FUNCTION_BLOCK "GCS7_E_PressureRange"	// FB 16
TITLE = PressureRange
//  
//COPYRIGHT:    (C) 1996  BUHLER AG, CH-9240 UZWIL, SWITZERLAND
//
//PRODUCT:      GCS7
//
//TITLE:        Pressure Range
//
//-------------------------------------------------------------------------
//
//IDENT:        AUTHOR:             DEPT:                       DATE:
//
//FB16.4.1      A. Egli             CT3                         09-Mar-2004
//              PCDirect Control: CmdReportOn,CmdReportOff=Bit14
//FB16.4.0      A. Egli             CT3                         17-Jun-2002
//              New Release with one block 
//FB16.2.2      S. Kalberer         CT3                         16-Oct-2000
//              LOG-entry corrected: SPN -> SPBN
//FB16.2.1      A. Egli             CT3                         08-Mai-2000
//              Local: StOverP --> StMinP
//              Set alarm horn by rising edge OutNoMinP
//FB16.2B       A. Egli             CT3                         23-Nov-1999
//              Message Nr StCtoOverP
//FB16.2A       A. Egli             CT3                         04-Mai-1998
//              StFault = StCode 32
//FB16.1A       S. Kalberer         AEE61                       10-Jul-1997
//              1st Release in S7
//
//-------------------------------------------------------------------------
//
//PURPOSE:      MANUAL : see [PRAENMAN]
//
//RESTRICTIONS: S7
//              ACCU2: Pointer to dynamic datas of the element
//              ACCU1: Pointer to parameter datas of the element
//
//-------------------------------------------------------------------------
//=======================================================
//Log Message: 
//------------------------------------------------------
// 0  normal pressure  
// 1  high pressure
// 2  over pressure
// 3  no minimum pressure
// 9  fault cancelled
// 10 fault
//
//=======================================================
//StCode:  State               
//------------------------------------------------------
//32  StFault             
// 1  StMinP              
//41  StMinP.HWStop       
//51  StMinP.DPFault      
// 3  StNormalP           
//43  StNormalP.HWStop    
//53  StNormalP.DPFault   
// 4  StCtoOverP          
//44  StCtoOverP.HWStop   
//54  StCtoOverP.DPFault  
// 5  StOverP             
//45  StOverP.HWStop      
//55  StOverP.DPFault     
// 6  StNormalP.Warning  
//
//
//
AUTHOR : EA
FAMILY : GCS7LL
NAME : PRang
VERSION : 4.1
VAR
  StCode : INT ;	//Element state code
  InMonMinP : BOOL ;	//Monitoring the minimum pressure
  spare0201 : BOOL ;
  spare0202 : BOOL ;
  spare0203 : BOOL ;
  spare0204 : BOOL ;
  spare0205 : BOOL ;
  InpMin : BOOL ;	//Digital input: Value <= min
  InpMax : BOOL ;	//Digital input: Value >= max
  spare0300 : BOOL ;
  spare0301 : BOOL ;
  spare0302 : BOOL ;
  CmdFaultReset : BOOL ;	//Command to reset fault
  InLocal : BOOL ;	//1= Local mode (no fault by Over Pressure)
  spare0305 : BOOL ;
  InReport : BOOL ;	//Report of all state transition
  spare0307 : BOOL ;
  InHWStop : BOOL ;	//HW stop is detected, no fault
  InDPFault : BOOL ;	//DP-Fault is detected, no fault
  OutNoMinP : BOOL ;	//Warning no minimum pressure
  spare0403 : BOOL ;
  spare0404 : BOOL ;
  spare0405 : BOOL ;
  spare0406 : BOOL ;
  spare0407 : BOOL ;
  StMinP : BOOL ;	//Value <= Minimum
  StNormalP : BOOL ;	//Value in Range Minimum to Maximum
  StOverP : BOOL ;	//Value >= Maximum (only in local mode)
  StCtoOverP : BOOL ;	//Value >= Maximum, delay time is active
  StFault : BOOL ;	//Element has a fault
  OutAlarmNrLog : INT ;	//Last textnumber send to log
  Par : STRUCT
   ParObjectNo : INT ;	//Is used for communication with PC, e.g. for message
   ParMsgType : INT ;	//Is used for message (translation of state)
   ParHornCode : INT ;	//Is used by horn module
   ParLogOff : BOOL ;	//Report is off
   ParDelayChange : INT ;	//t0, maximum time until state changes to StCtoOverP
   ParDelayMin : INT ;	//t1, maximum time until state changes to StMinP
   ParDelayMax : INT ;	//t2, maximum time until state changes to StOverP or StFault
   ParMonMinP : INT ;	//t3, if InMonMinP: maximum time to be out of MinP until OutNoMinP
   OutMonTime : INT ;	//Actual value monitoring time t3
   OutDelayMinTime : INT ;	//Actual value delay time t1
   OutDelayMaxTime : INT ;	//Actual value delay time t0,t2
  END_STRUCT ;
END_VAR
VAR_TEMP
  tmpLOGvalue : WORD ;	//LOG value
  tmpLenDyn : DINT ;
  tmpReport : BOOL ;	//Global LOG all
  tmpDelayOver : BOOL ;	//Delay time is over
  tmpLocal : BOOL ;
END_VAR
BEGIN
NETWORK
TITLE =  Start Global
      L     30;
      T     #tmpLenDyn;	// Length Dynamic datas
NETWORK
TITLE = PC Control
//=== Test Object number =====================
      L     "SYS_DirectCtrlDB".PC.ObjectNo;	//PCControl.ObjectNo
      L     #Par.ParObjectNo;	//Input ObjectNo
      <>I;
      JC    Ctrl;
//=== Test OType      ========================
      L     1016;	//Input object type
      L     "SYS_DirectCtrlDB".PC.ObjectType;	//PCControl.ObjectType
      <>I;
      JC    Ctrl;
//=== Test Handshake =========================
      A     "SYS_DirectCtrlDB".PC.Hsk.FExamine;	// Handshake.FExamine
      JC    pExa;
      A     "SYS_DirectCtrlDB".PC.Hsk.FDefineCmd;	// Handshake.FDefineCmd
      JC    pCmd;
      A     "SYS_DirectCtrlDB".PC.Hsk.FDefinePara;	// Handshake.FDefinePara
      JC    pPar;
pIni: L     2;	// FcInit
      UC    "SYS_DirectCtrl";
      JU    Ctrl;
// Write parameter 
pPar: LAR1  P#DBX 58.0;
      L     P##Par;
      L     DW#16#FFFFF;
      AD;
      +AR1;
      L     DBW [AR1,P#8.0];
      T     #Par.ParDelayChange;
      L     DBW [AR1,P#10.0];
      T     #Par.ParDelayMin;
      L     DBW [AR1,P#12.0];
      T     #Par.ParDelayMax;
      L     DBW [AR1,P#14.0];
      T     #Par.ParMonMinP;
// Write new commands from PC to Interface object
pCmd: A     "SYS_DirectCtrlDB".PC.Cmd1[11];	// CmdFaultReset
      S     #CmdFaultReset;
      A     "SYS_DirectCtrlDB".PC.Cmd1[14];	// CmdReportOn    [4.1]
      S     #InReport;
      A     "SYS_DirectCtrlDB".PC.Cmd2[14];	// CmdReportOff   [4.1]
      R     #InReport;
      JU    pIni;
pExa: TAR2;	// Address Dynamic datas
      T     "SYS_DirectCtrlDB".GC.InDynAddr;	// -->PCControl.GC.InDynAddr
      L     #tmpLenDyn;	// Length Dynamic datas
      T     "SYS_DirectCtrlDB".GC.InDynLen;	// -->PCControl.GC.InDynLen
      L     0;
      T     "SYS_DirectCtrlDB".GC.InParaAddr;	// -->PCControl.GC.InParaAddr
      T     "SYS_DirectCtrlDB".GC.InParaLen;	// -->PCControl.GC.InParaLen
      L     1;	// Code FcExamine
      UC    "SYS_DirectCtrl";
      L     10;	//Revision
      T     "SYS_DirectCtrlDB".GC.Revision;
NETWORK
TITLE =  All State Init
//===Global Group Orders===
//---Report is on---
Ctrl: O     "GCS7_Gr_OutReportAll";	//---Global OutReportAll
      O     #InReport;
      =     #tmpReport;
      A     #InLocal;
      O     #InHWStop;
      O     #InDPFault;
      =     #tmpLocal;
// Monitoring
//---Condition to start monitoring time:  Monitoring is on
      A     #InMonMinP;
      AN    #StMinP;	// State minimum pressure
      JC    MO2;
      R     #OutNoMinP;
      L     #Par.ParMonMinP;	// Set monitoring time
      T     #Par.OutMonTime;
      JU    STAT;
//---Condition for monitoring
MO2:  A     #OutNoMinP;	// Monitoring output
      JC    STAT;
      AN    "GCS7_Gr_OutTick200ms";	//Gr.OutTick200ms
      L     #Par.OutMonTime;
      JC    MO3;
      +     -2;	// Decrement all 200ms
      T     #Par.OutMonTime;
MO3:  L     0;
      >I;	// Check monitoring time t3 over
      JC    STAT;
      S     #OutNoMinP;	// set monitoring output
      S     "GCS7_Gr_InFaultFlag";	// InFaultFlag
      CALL  "SYS_Horn_Code" (
           FcCode                   := 1,
           ParObjectType            := 1016,
           ParObjectNo              := #Par.ParObjectNo,
           ParHornCode              := #Par.ParHornCode);
      JU    LOG3;
NETWORK
TITLE = States
STAT: A     #StMinP;	//===State machine===
      JC    MP;
      A     #StNormalP;
      JC    NP;
      A     #StCtoOverP;
      JC    COP;
      A     #StOverP;
      JC    OP;
      A     #StFault;
      JC    FLT;
      S     #StMinP;	//Initialise: goto StMinP
NETWORK
TITLE = StMinP
MP:   A     #InpMin;	//---Condition for StMinP
      AN    #InpMax;
      JC    SAVE;
      R     #StMinP;	//---Transition --> StNormal
      S     #StNormalP;
      L     #Par.ParDelayChange;
      T     #Par.OutDelayMaxTime;
      JU    LOG1;
NETWORK
TITLE = StNormalP
//Logic
//---Condition for StCtoOverP
NP:   A     #InpMax;
      JC    NPJ1;
      L     #Par.ParDelayChange;
      T     #Par.OutDelayMaxTime;
//---Condition for StNormalP
      A     #InpMin;
      R     #StNormalP;
      S     #StMinP;
      JU    SAVE;
NPJ1: L     #Par.OutDelayMaxTime;
      AN    "GCS7_Gr_OutTick200ms";	//Gr.OutTick200ms
      JC    NPJ2;
      +     -2;	// Decrement all 0.2s
      T     #Par.OutDelayMaxTime;
NPJ2: L     0;
      >I;
      JC    SAVE;
//---Transition --> StCtoOverP
      R     #StNormalP;
      S     #StCtoOverP;
      L     #Par.ParDelayMax;
      T     #Par.OutDelayMaxTime;
      L     #Par.ParDelayMin;
      T     #Par.OutDelayMinTime;
      JU    LOG1;
NETWORK
TITLE = StCtoOverP
//---Condition for StCtoOverP
COP:  AN    "GCS7_Gr_OutTick200ms";	//Gr.OutTick200ms
      L     #Par.OutDelayMaxTime;
      JC    COP1;
      +     -2;	// Decrement all 0.2s
      T     #Par.OutDelayMaxTime;
COP1: L     0;
      >I;
      JC    COPM;
//---Transition --> StFault
      AN    #tmpLocal;
      R     #StCtoOverP;
      JC    xxS4;
//---Transition --> StOverP
      R     #StCtoOverP;
      S     #StOverP;
      JU    LOG1;
//---Condition for StMinP
//Condition delay time minimum
COPM: A     #InpMin;
      AN    #InpMax;
      JC    COP6;
      L     #Par.ParDelayMin;
      T     #Par.OutDelayMinTime;
      JU    SAVE;
COP6: AN    "GCS7_Gr_OutTick200ms";	//Gr.OutTick200ms
      L     #Par.OutDelayMinTime;
      JC    COP7;
      +     -2;	// Decrement all 0.2s
      T     #Par.OutDelayMinTime;
COP7: L     0;
      >I;
      JC    SAVE;
//---Transition --> StMinP
      R     #StCtoOverP;
      S     #StMinP;
      JU    LOG1;
NETWORK
TITLE = StOverP
OP:   AN    #InpMin;	//---Condition for StOverP
      O     #InpMax;
      A     #tmpLocal;
      JC    SAVE;
      A     #InpMin;	//---Condition for StMinP
      AN    #InpMax;
      JC    OP5;
      R     #StOverP;	//---Transition --> StFault
      JU    xxS4;
OP5:  R     #StOverP;	//---Transition --> StMinP
      S     #StMinP;
      JU    LOG1;
NETWORK
TITLE = StFault
// Any transiton to Fault  
xxS4: SET;
      S     #StFault;
      S     "GCS7_Gr_InFaultFlag";	// InFaultFlag
      CALL  "SYS_Horn_Code" (
           FcCode                   := 1,
           ParObjectType            := 1016,
           ParObjectNo              := #Par.ParObjectNo,
           ParHornCode              := #Par.ParHornCode);
      JU    LOG8;
//===logic
FLT:  AN    "GCS7_Gr_OutFaultReset";	//---Condition for StFault
      AN    #CmdFaultReset;
      AN    #InLocal;
      JC    SAVE;
      AN    #InpMin;	//---reLOG Fault
      O     #InpMax;
      AN    #tmpLocal;
      JC    LOG8;
      AN    #InpMin;	//---Condition for StOverP
      O     #InpMax;
      A     #tmpLocal;
      JC    FLT8;
      R     #StFault;	//---Transition --> StMinP
      S     #StMinP;
      JU    LOG9;
FLT8: R     #StFault;	//---Transition --> StOverP
      S     #StOverP;
      JU    LOG9;
NETWORK
TITLE = LOG Message
LOG1: AN    #tmpReport;	//---Report all?
      JC    SAVE;	// [2.2]
      A     #StMinP;
      O     #StNormalP;
      L     B#(4, 0);	//Message Class Information normal pressure
      JC    LOG;
      A     #StCtoOverP;
      L     B#(4, 1);	// Message Class Information high pressure
      JC    LOG;
      A     #StOverP;
      L     B#(4, 2);	// Message Class Information over pressure [Rel2B]
      JC    LOG;
      JU    SAVE;
LOG3: L     B#(4, 3);	// Message Class Information no minimum pressure reached
      JU    LOG;
LOG8: L     B#(1, 10);	// Message Class Error Message
      JU    LOG;
LOG9: L     B#(3, 9);	// Message Class Operate fault cancelled
LOG:  A     #Par.ParLogOff;	//---Set LOG Message
      JC    SAVE;
      T     #tmpLOGvalue;
      L     W#16#FF;
      AW;
      T     #OutAlarmNrLog;
      CALL  "GCS7_LogConvert" (
           ObjectNo                 := #Par.ParObjectNo,
           MsgType                  := #Par.ParMsgType,
           ClassMsgTxt              := #tmpLOGvalue,
           OType                    := 1016);	// LOG Message Converter / Entry / Contains Class and TextNo
NETWORK
TITLE = Global End
SAVE: CLR;	//---Clear all commands
      =     #CmdFaultReset;
//--Output for group 
      A     #InDPFault;
      AN    #InLocal;
      S     "GCS7_Gr_InDPFault";
      A     #InHWStop;
      AN    #InLocal;
      S     "GCS7_Gr_InHWStop";
NETWORK
TITLE = State Code
      A     #StMinP;
      L     1;	// Code: minimum
      JC    STC8;
      A     #StNormalP;
      A     #OutNoMinP;
      AN    #tmpLocal;
      L     6;	// Code: normal.warning
      JC    STC8;
      A     #StNormalP;
      L     3;	// Code: normal.ok
      JC    STC8;
      A     #StCtoOverP;
      L     4;	// Code: high
      JC    STC8;
      A     #StOverP;
      L     5;	// Code: over
      JC    STC8;
      JU    STCF;
STC8: AN    #InHWStop;
      JC    STCD;
      +     40;	//StXxx.HWStop
      JU    STC9;
STCD: AN    #InDPFault;
      JC    STC9;
      +     50;	//StXxx.DPFault
      JU    STC9;
STCF: L     32;	// Code: fault
STC9: L     #StCode;	// Old state code
      TAK;
      T     #StCode;	// Save state code
      <>I;
      L     3;	// Load code for CBit methode
      CC    "SYS_CBitCtrl";
END_FUNCTION_BLOCK

FUNCTION_BLOCK "GCS7_E_AnalogOutput"	// FB 17
TITLE = Analog Output
//  
//COPYRIGHT:    (C) 1997 BY  BUHLER LTD.
//                           CH-9240 UZWIL  SWITZERLAND
//
//PRODUCT:      GCS7
//
//TITLE:        Element Analog Output
//
//-------------------------------------------------------------------------
//
//IDENT:        AUTHOR:             DEPT:                       DATE:
//
//FB17.3.2      A. Egli             CT3                         19-Dec-2007
//              StFault->StOff Check InManual 
//FB17.3.1      A. Egli             CT3                         04-Aug-2003
//              -Read M12.3 "GCS7_Gr_OutFaultReset"   
//FB17.3.0      A. Egli             CT3                         17-Jun-2002
//              -New Release with one block 
//              -OutpFaultReset
//              -ParFU
//FB17.2.1      A. Egli             CT3                         18-Mai-2001
//              Calculation Output, if ParUnitsByZeroDigit >0
//FB17.2A       A. Egli             CT3                         04-Mai-1998
//              StFault = StCode 32
//FB17.1A       S. Kalberer         AEE61                       16-Jul-1997
//              1st Release in S7
//
//-------------------------------------------------------------------------
//
//PURPOSE:      MANUAL : see [AOxxMAN]
//
//RESTRICTIONS: S7
//              ACCU2: Pointer to dynamic datas of the element
//              ACCU1: Pointer to parameter datas of the element
//
//-------------------------------------------------------------------------
//
//MaxDigits:     Siemens: 27'648/ Wago: 32'767
//
//=======================================================
//Log Message: 
//-------------------------------------------------------
// 0  off
// 2  on
// 9  fault cancelled
//10  fault device
//
//=======================================================
//StCode:  State               
//------------------------------------------------------
//32  StFault        
// 1  StOff          
//41  StOff.HWStop    
//51  StOff.DPFault   
//61  StOff.FaultDev   (Passiv)
// 3  StOn           
//
AUTHOR : EA
FAMILY : GCS7LL
NAME : AO
VERSION : 3.2
VAR
  StCode : INT ;	//Element state code
  InDisable : BOOL ;	//Disable the output, set OutValue to zero.
  spare0201 : BOOL ;
  spare0202 : BOOL ;
  spare0203 : BOOL ;
  spare0204 : BOOL ;
  spare0205 : BOOL ;
  spare0206 : BOOL ;
  InpFaultDev : BOOL ;	//Digital input: 1= overload or fault frequency converter
  spare0300 : BOOL ;
  spare0301 : BOOL ;
  spare0302 : BOOL ;
  CmdFaultReset : BOOL ;	//Command to reset fault
  InLocal : BOOL ;	//Local mode
  InManual : BOOL ;	//1= Manual/ 0=Automatic
  InReport : BOOL ;	//Report all state transitions
  spare0307 : BOOL ;
  InHWStop : BOOL ;	//HW stop is detected, no fault
  InDPFault : BOOL ;	//DP-Fault is detected, no fault
  spare0402 : BOOL ;
  spare0403 : BOOL ;
  spare0404 : BOOL ;
  OutpFaultReset : BOOL ;	//Reset Alarm
  OutMin : BOOL ;	//Signal OutValue <= ParLimitMin
  OutMax : BOOL ;	//Signal OutValue >= ParLimitMax
  StOff : BOOL ;	//Analog output is disabled
  spare0501 : BOOL ;
  StOn : BOOL ;	//Analog output is on
  spare0503 : BOOL ;
  StFault : BOOL ;	//Fault device was detected
  OutpValue : INT ;	//Converted value to set analog output
  InOutValuePc : INT ;	//Set value in percent
  InOutValueUnits : DINT ;	//Set value in units
  ASW : DINT ;	//Free for user software
  OutAlarmNrLog : INT ;	//Last textnumber send to log
  Par : STRUCT
   ParObjectNo : INT ;	//Is used for communication with PC, e.g. for message
   ParMsgType : INT ;	//Is used for message (translation of state)
   ParHornCode : INT ;	//Is used by horn module
   ParLogOff : BOOL ;	//Report is off
   ParFU : BOOL ;	//FU, 0% = 0%Digits =ParUnitsByZeroDigit
   ParValuePc : BOOL ;	//InOutValue specification in percent not in units.
   ParLimitsPc : BOOL ;	//Limits in percent not in units
   ParWago : BOOL ;	//Wago analog output module format
   ParUnitsByZeroDigit : DINT ;	//Value in units by analog signal=0
   ParUnitsByMaxDigit : DINT ;	//Value in units by maximum analog signal
   ParUnitsBy100Pc : DINT ;	//Value in units by 100% of InOutValuePc
   ParLimitMin : DINT ;	//Minimum limit: value in units or percent
   ParLimitMax : DINT  := L#10000;	//Maximum limit: value in units or percent
   ParDelayTime : INT ;	//Requested fault delay time by InpFaultDev
   OutDelayTime : INT ;	//Actual time: DelayTime
  END_STRUCT ;
END_VAR
VAR_TEMP
  tmpLenDyn : DINT ;
  tmpLOGvalue : WORD ;	//LOG value
  tmpDConverter : REAL ;	//provisional result: ParUnitsByMaxDigit - ParUnitsByZeroDigit
  tmpOutValueUnits : REAL ;	//Limited value
  tmpFaultDelayDone : BOOL ;
  tmpLocal : BOOL ;
  tmpValueDiff : REAL ;
  tmpValueZero : REAL ;
END_VAR
BEGIN
NETWORK
TITLE = Start Global
      L     52;
      T     #tmpLenDyn;	//--> Len dynamic data in byte
NETWORK
TITLE = PC Control
      L     "SYS_DirectCtrlDB".PC.ObjectNo;	//PCControl.ObjectNo
      L     #Par.ParObjectNo;	//Input ObjectNo
      <>I;
      JC    Ctrl;
//=== Test OType      ========================
      L     1017;	//Input object type
      L     "SYS_DirectCtrlDB".PC.ObjectType;	//PCControl.ObjectType
      <>I;
      JC    Ctrl;
//!!!=== Address definition !!!! =============
//=== Test Handshake =========================
      A     "SYS_DirectCtrlDB".PC.Hsk.FExamine;	// PC.Hsk.FExamine
      JC    pExa;
      A     "SYS_DirectCtrlDB".PC.Hsk.FDefineCmd;	// PC.Hsk.FDefineCmd
      O     "SYS_DirectCtrlDB".PC.Hsk.FDefineValue;	// PC.Hsk.FDefineValue
      JC    pCmd;
      A     "SYS_DirectCtrlDB".PC.Hsk.FDefinePara;	// PC.Hsk.FDefinePara
      JC    pPar;
pIni: L     2;	// FcInit
      UC    "SYS_DirectCtrl";
      JU    Ctrl;
// Write parameter 
pPar: LAR1  P#DBX 58.0;
      L     P##Par;
      L     DW#16#FFFFF;
      AD;
      +AR1;
      L     DBD [AR1,P#20.0];
      T     #Par.ParLimitMin;
      L     DBD [AR1,P#24.0];
      T     #Par.ParLimitMax;
      L     DBW [AR1,P#28.0];
      T     #Par.ParDelayTime;
// Write new commands from PC to Interface object
pCmd: A     "SYS_DirectCtrlDB".PC.Cmd1[0];	//Cmd1[0]= CmdDisableOn
      S     #InDisable;
      A     "SYS_DirectCtrlDB".PC.Cmd2[0];	//Cmd2[0]= CmdDisableOff
      R     #InDisable;
      A     "SYS_DirectCtrlDB".PC.Cmd1[11];	//Cmd1[11]= CmdFaultReset
      S     #CmdFaultReset;
      A     "SYS_DirectCtrlDB".PC.Cmd1[14];	//Cmd1[14]= CmdReportOn
      S     #InReport;
      A     "SYS_DirectCtrlDB".PC.Cmd2[14];	//Cmd2[14]= CmdReportOff
      R     #InReport;
      A     "SYS_DirectCtrlDB".PC.Cmd1[13];	// CmdManualOn
      S     #InManual;
      A     "SYS_DirectCtrlDB".PC.Cmd2[13];	// CmdManualOff
      O     "GCS7_Gr_OutManualOff";	//Global.OutManualOff  [2.10]
      R     #InManual;
//Define Value
      AN    "SYS_DirectCtrlDB".PC.Hsk.FDefineValue;	// PC.Hsk.FDefineValue
      ON    #InManual;
      JC    pIni;
      LAR1  P#DBX 58.0;
      L     DBD [AR1,P#10.0];
      T     #InOutValueUnits;
      JU    pIni;
pExa: TAR2;	// Address Dynamic datas
      T     "SYS_DirectCtrlDB".GC.InDynAddr;	// -->PCControl.GC.InDynAddr
      L     #tmpLenDyn;	// Length Dynamic datas
      T     "SYS_DirectCtrlDB".GC.InDynLen;	// -->PCControl.GC.InDynLen
      L     0;
      T     "SYS_DirectCtrlDB".GC.InParaAddr;	// -->PCControl.GC.InParaAddr
      T     "SYS_DirectCtrlDB".GC.InParaLen;	// -->PCControl.GC.InParaLen
      L     1;	// Code FcExamine
      UC    "SYS_DirectCtrl";
      L     10;	//Revision
      T     "SYS_DirectCtrlDB".GC.Revision;
Ctrl: NOP   0;
NETWORK
TITLE = Init
//Manual Mode
      A     "GCS7_Gr_OutManualOff";	//GCS7_Gr_OutManualOff
      R     #InManual;
      A     #InManual;
      S     "GCS7_Gr_InManual";	//GCS7_Gr_InManual
//Local
      A     #InLocal;
      AN    #InManual;
      O     #InHWStop;
      O     #InDPFault;
      =     #tmpLocal;
NETWORK
TITLE = Calculate InOutValuePc or InOutValueUnits : ParFU=1
      A     #Par.ParFU;
      JC    c1En;
//--Calculate the other InOutValue
      A     #Par.ParValuePc;
      JC    c1PC;
//---InOutValuePc
      L     #InOutValueUnits;
      DTR;
      T     #tmpOutValueUnits;
      L     #Par.ParUnitsBy100Pc;
      DTR;
      /R;	//    InOutValueUnits
      L     1.000000e+04;	// = ----------------  * 10'000
      *R;	//    ParUnitsBy100Pc 
      RND;
      T     #InOutValuePc;
      JU    c1En;
//---InOutValueUnits
c1PC: L     #InOutValuePc;
      ITD;
      DTR;
      L     1.000000e+04;
      /R;
      L     #Par.ParUnitsBy100Pc;	//   InOutValuePc
      DTR;	// = ------------ * ParUnitsBy100Pc       
      *R;	//      10'000
      T     #tmpOutValueUnits;
      RND;
      T     #InOutValueUnits;	//-->Digits
c1En: NOP   0;
NETWORK
TITLE = Calculate InOutValuePc or InOutValueUnits: ParFU=1
      AN    #Par.ParFU;
      JC    fuEn;
      L     #Par.ParUnitsBy100Pc;	// 
      DTR;	//       
      L     #Par.ParUnitsByZeroDigit;	// 
      DTR;	//       
      T     #tmpValueZero;
      -R;
      T     #tmpValueDiff;
//--Calculate the other InOutValue
      A     #Par.ParValuePc;
      JC    fuPC;
//---InOutValuePc
      L     #InOutValueUnits;
      DTR;
      T     #tmpOutValueUnits;
      L     #tmpValueZero;
      -R;
      L     #tmpValueDiff;
      /R;	//    InOutValueUnits-ParUnitsByZeroDigit
      L     1.000000e+04;	// = ------------------------------------  * 10'000
      *R;	//    ParUnitsBy100Pc-ParUnitsByZeroDigit 
      RND;
      T     #InOutValuePc;
      JU    fuEn;
//---InOutValueUnits
fuPC: L     #InOutValuePc;
      ITD;
      DTR;
      L     1.000000e+04;
      /R;
      L     #tmpValueDiff;	//   InOutValuePc
      *R;	// = ------------ * (ParUnitsBy100Pc-ParUnitsByZeroDigit) +ParUnitsByZeroDigit     
      L     #tmpValueZero;	//      10'000
      +R;
      T     #tmpOutValueUnits;
      RND;
      T     #InOutValueUnits;	//-->Digits
fuEn: NOP   0;
NETWORK
TITLE = Test limits
//--Test limits---
      A     #Par.ParLimitsPc;	// Limit in percent
      JC    LiPc;
      L     #InOutValueUnits;
      L     #Par.ParLimitMax;	// Calculation limit maximum
      >D;
      =     #OutMax;
      R     #OutMin;
      JC    Lmax;	// --> Limit max
      L     #InOutValueUnits;
      L     #Par.ParLimitMin;	// Calculation limit minimum
      <D;
      =     #OutMin;
      JCN   LiEn;
Lmax: DTR;
      T     #tmpOutValueUnits;
      JU    LiEn;
//-- Limits in procent 
LiPc: L     #InOutValuePc;
      ITD;
      L     #Par.ParLimitMax;	// Calculation limit maximum
      >=D;
      =     #OutMax;
      R     #OutMin;
      JC    L2mx;
      TAK;
      L     #Par.ParLimitMin;	// Calculation limit minimum
      <=D;
      =     #OutMin;
      JCN   LiEn;
L2mx: DTR;
      L     1.000000e+04;
      /R;
      L     #Par.ParUnitsBy100Pc;	//---Calculate provisional result: tmpDProcess
      DTR;
      *R;
      T     #tmpOutValueUnits;
LiEn: NOP   0;
NETWORK
TITLE = Fault delay time: ParDelayTime 
//Test or Running delay time ====================
//---Condition for Delay Fault
      A     #InpFaultDev;
      JC    TFF1;
      R     #tmpFaultDelayDone;
      L     0;
      T     #Par.OutDelayTime;
      JU    TFF0;
TFF1: AN    "GCS7_Gr_OutTick200ms";	// Decrement all 200ms
      L     #Par.OutDelayTime;
      JC    TFF3;
      +     2;
TFF3: T     #Par.OutDelayTime;
      L     #Par.ParDelayTime;
      >=I;
      =     #tmpFaultDelayDone;
      JCN   TFF0;
      T     #Par.OutDelayTime;
TFF0: NOP   0;
NETWORK
TITLE = States
      A     #StOn;
      JC    S2;
      A     #StOff;
      JC    S0;
      A     #StFault;
      JC    S4;
      S     #StOn;	//Initialise: goto StOn
      JU    S2;
NETWORK
TITLE = StOff
// Any transiton to StOff  
xxS0: SET;
      S     #StOff;
      L     B#(4, 0);	// MessageClass Info "Off"
      JU    REPO;
//---- Logic ---
//Transition to StFault
S0:   A     #tmpFaultDelayDone;
      AN    #tmpLocal;
      R     #StOff;
      JC    xxS4;	//-->StFault  
      A     #InDisable;
      O     #tmpLocal;
      JC    OUT;
//Transition to StOn
      R     #StOff;
      JU    xxS2;	//-->StOn
NETWORK
TITLE = StOn
// Any transiton to StOff  
xxS2: SET;
      S     #StOn;
      L     B#(4, 2);	// MessageClass Info "On"
      JU    REPO;
//---- Logic ---
//Transition to StFault
S2:   A     #tmpFaultDelayDone;
      AN    #tmpLocal;
      R     #StOn;
      JC    xxS4;	//---> StFault
//Transition to StOff
      A     #InDisable;
      O     #tmpLocal;
      R     #StOn;
      JC    xxS0;	//---> StOff
      JU    OUT;
NETWORK
TITLE = StFault
// Any transiton to Fault  
xxS4: SET;
      S     #StFault;
      S     "GCS7_Gr_InFaultFlag";	//Gr.InFaultFlag
      CALL  "SYS_Horn_Code" (
           FcCode                   := 1,
           ParObjectType            := 1017,
           ParObjectNo              := #Par.ParObjectNo,
           ParHornCode              := #Par.ParHornCode);
S4MG: L     B#(1, 10);	// MessageClass Error "fault device"
      JU    LOG;
//==Logic====
S4:   A     #InLocal;
      AN    #InManual;	//[3.2]
      JC    S4xx;
//-Wait for fault reset
      AN    "GCS7_Gr_OutTick500ms";	// Gr.OutTick500ms //[3.0]
      ON    #OutpFaultReset;	//                   [3.0]
      JC    OUT;	//                   [3.0]
      R     #OutpFaultReset;	//                   [3.0]
      A     #InpFaultDev;
      AN    #tmpLocal;
      JC    S4MG;	//--> Retry Message
// Transition to StOff;
S4xx: R     #StFault;
      S     #StOff;
      L     B#(3, 9);	// MessageClass Operater "fault cancelled"
      JU    LOG;
NETWORK
TITLE = LOG Message
REPO: AN    #InReport;
      AN    "GCS7_Gr_OutReportAll";	//---Gr.OutReportAll
      JC    OUT;
LOG:  A     #Par.ParLogOff;	//---Set LOG Message
      JC    OUT;
      T     #tmpLOGvalue;
      L     W#16#FF;
      AW;
      T     #OutAlarmNrLog;
      CALL  "GCS7_LogConvert" (
           ObjectNo                 := #Par.ParObjectNo,
           MsgType                  := #Par.ParMsgType,
           ClassMsgTxt              := #tmpLOGvalue,
           OType                    := 1017);	// LOG Message Converter / Entry / Contains Class and TextNo
NETWORK
TITLE = Global End
OUT:  NOP   0;
      A     "GCS7_Gr_OutFaultReset";	// Gr.OutFaultReset
      S     #CmdFaultReset;
//===Set Output fault reset
      A     "GCS7_Gr_OutTick500ms";	// Gr.OutTick500ms
      AN    #StFault;
      R     #OutpFaultReset;
//===OutpFaultReset
      A     "GCS7_Gr_OutTick500ms";	// Gr.OutTick500ms
      A     #CmdFaultReset;
      S     #OutpFaultReset;
      R     #CmdFaultReset;
//--Output for group 
      A     #InDPFault;
      AN    #InLocal;
      S     "GCS7_Gr_InDPFault";
      A     #InHWStop;
      AN    #InLocal;
      S     "GCS7_Gr_InHWStop";
NETWORK
TITLE =  Calculate analog output
      A     #StOn;
      JC    aoJ1;	//--> Set to 0
      L     #Par.ParUnitsByZeroDigit;	//[2.1]
      DTR;
      T     #tmpOutValueUnits;
aoJ1: L     #Par.ParUnitsByMaxDigit;
      L     #Par.ParUnitsByZeroDigit;
      -D;
      DTR;
      T     #tmpDConverter;
      L     #tmpOutValueUnits;
      L     #Par.ParUnitsByZeroDigit;
      DTR;	//        (InOutValueUnits    - ParUnitsByZeroDigit)
      -R;	// ==  ------------------------------------------ * MaxDigits
      L     #tmpDConverter;	//        (ParUnitsByMaxDigit - ParUnitsByZeroDigit)
      /R;
      L     3.276700e+04;	//MaxDigits for Wago
      A     #Par.ParWago;
      JC    aoJ2;
      TAK;
      L     2.764800e+04;	//MaxDigits for Siemens
aoJ2: *R;
      RND;
      T     #OutpValue;	//--> Analog output value
//---Limit OutpValue if calculated output value >32'767 or <-32'768 to max. value
      L     L#32767;
      <=D;
      JC    aoJ3;
      T     #OutpValue;
      JU    aoJ9;
aoJ3: TAK;
      L     L#-32768;
      >=D;
      JC    aoJ9;
      T     #OutpValue;
aoJ9: NOP   0;
NETWORK
TITLE = State Code
      AN    #StOff;
      JC    STC2;
      L     41;	//Code: StOff.HWStop
      A     #InHWStop;
      JC    STC9;
      L     51;	//Code: StOff.DPFault
      A     #InDPFault;
      JC    STC9;
      A     #InpFaultDev;	//Code: StOff.InpFaultDev
      L     61;
      JC    STC9;
      L     1;	// Code: stopped
      JC    STC9;
//--------------------
STC2: L     3;	// Code: on
      A     #StOn;
      JC    STC9;
//--------------------
      L     32;	// Code: fault
STC9: L     #StCode;	// Old state code
      TAK;
      T     #StCode;	// Save state code
      <>I;
      L     3;	// Load code for CBit methode
      CC    "SYS_CBitCtrl";
END_FUNCTION_BLOCK

FUNCTION_BLOCK "GCS7_E_ATV"	// FB 18
TITLE = ATV
//
//COPYRIGHT:    (C) 2006  BUHLER AG, CH-9240 UZWIL, SWITZERLAND
//
//PRODUCT:      GCS7
//
//TITLE:        FU Control Altivar
//
//REVISION:     10
//-------------------------------------------------------------------------
//
//IDENT:        AUTHOR:             DEPT:                       DATE:
//FB18.1.8      Ph.Engler           GP92                        05-Jun-2009
//              - Calculation of OutSpeed depending of ParValueAsUnit
//FB18.1.7      A. Egli             BASE                        16-Mai-2008
//              Text-No 96: Fault Communication
//FB18.1.6      A. Egli             BASE                        23-Apr-2008
//              - Run Delay time after CmdFaultReset
//FB18.1.5      A. Egli             BASE                        07-Apr-2008
//              - NMAx data from FU copied to data block
//              - CmdFaultReset from Group
//FB18.1.3      A. Egli             CT3                         18-Apr-2007
//              Multimotor configuration
//FB18.1.1      A. Egli             CT3                         24-Nov-2006
//              Local Mode: Condition StStooping-->StStarting
//FB18.1.0      A. Egli             CT3                         26-Sep-2006
//              1st Release in S7
//
//-------------------------------------------------------------------------
//
//PURPOSE:      MANUAL : see [SSW-EL--Altivar_MAN_en]
//
//RESTRICTIONS: S7
//-------------------------------------------------------------------------
//
//
//=======================================================
//Log Message: 
//------------------------------------------------------
// 0  stopped
// 2  started forward
// 5  started reverse
// 9  fault cancelled
//10  fault device
//11  fault running
//12  fault starting
//13  fault stopping
//14  fault Isolated
//15  fault Overload
//16  fault Service
//
//=======================================================
//StCode:  State               
//------------------------------------------------------
// 1 StStopped                 
// 2 StStarting                
// 3 StStartedFwdSlow          
// 4 StStartedFwdFast          
// 5 StStartedRevSlow          
// 6 StStartedRevFast          
// 7 StStopping                 
// 9 StStartRequest            StStopped+CmdNext 
//11 StartingDelay             StStopped+(OutStartWarning or OutStartDelay)
//
//31 StFault+InpFaultDev=1     (Active)
//32 StFault
//33 StFault+Isolated
//34 StFault+Overload
//35 StFault+Service 
AUTHOR : EA
FAMILY : GCS7LL
NAME : FU_ALT
VERSION : 1.8
VAR
  StCode : INT ;	//Element state code
  InEnableRev : BOOL ;	//Enable to run the element reverse
  InEnableFwd : BOOL ;	//Enable to run the element forward
  InPrestart : BOOL ;
  spare23 : BOOL ;
  spare24 : BOOL ;
  spare25 : BOOL ;
  InpContactor : BOOL ;
  spare27 : BOOL ;
  CmdOff : BOOL ;	//Pulse to stop the element immediately (manual mode)
  CmdOn : BOOL ;	//Pulse to start the element immediately (manual mode)
  CmdNext : BOOL ;	//Pulse to start the element in automatic mode (see global flags)
  CmdFaultReset : BOOL ;	//Command to reset fault
  InLocal : BOOL ;	//1= Local mode (no fault by start with service switch)
  InManual : BOOL ;	//1= Manual/ 0=Automatic
  InReport : BOOL ;	//Report of all state transitions
  InSeqStop : BOOL ;	//Stop automatically after idling time
  InHWStop : BOOL ;	//HW stop is detected, no fault
  InDPFault : BOOL ;	//DP-Fault is detected, no fault
  InSimulation : BOOL ;	//Simulation with DPSim
  OutIdling : BOOL ;	//Idling is active
  OutComFaultRead : BOOL ;
  OutComFaultWrite : BOOL ;
  OutpContactor : BOOL ;
  Spare47 : BOOL ;
  StStopped : BOOL ;	//Element is stopped
  StStarting : BOOL ;	//Element is starting
  StStartedFwd : BOOL ;	//Element is started forward: Next element can start
  StStopping : BOOL ;	//Element is stopping
  StFault : BOOL ;	//Element has a fault
  StStartedRev : BOOL ;	//Element is started reverse: Next Element can start
  InOutManRev : BOOL ;	//Manual direction mode: 1= reverse / 0= forward
  Spare57 : BOOL ;
  InForce : BOOL ;
  tmpASW : BOOL ;
  InpIsolated : BOOL ;
  InpOverload : BOOL ;
  InpService : BOOL ;
  InMultiMotorCfg0 : BOOL ;	//Use Multimotor configuration 0
  InMultiMotorCfg1 : BOOL ;	//Use Multimotor configuration 1
  InMultiMotorCfg2 : BOOL ;	//Use Multimotor configuration 2
  OutFaultRelevant : BOOL ;	//Relavant faultfor group
  OutDPFault : BOOL ;	//DP-Fault is detected, no fault
  OutStartRequestMan : BOOL ;	//Start Request for Manaul Mode
  OutStartRequestAuto : BOOL ;
  OutStartWarning : BOOL ;	//Startwarning is active
  OutStartDelay : BOOL ;	//Startdelay time is running
  OutDelayFault : BOOL ;	//ParDelayFaultTime is running
  OutAlarmNoLog : INT ;	//Last textnumber send to log
  OutFaultDev : BOOL ;	//Alarm reason
  OutFaultStopping : BOOL ;	//Alarm reason
  OutFaultStarting : BOOL ;	//Alarm reason
  OutFaultOverload : BOOL ;	//Alarm reason
  OutFaultIsolated : BOOL ;	//Alarm reason
  OutFaultService : BOOL ;	//Alarm reason
  OutTimeStarted : DINT ;	//[s] Not errasable time "Started"
  OutTimeFaulted : DINT ;	//[s] Not errasable time "Faulted"
  OutCntStartup : DINT ;	//Not errasable counter of startup
  OutCntFault : DINT ;	//Not errasable counter of faults
  InSpeed : REAL ;	//Target Value speed [Unit or 0.1%]
  OutSpeed : REAL ;	//Actual Value speed [0.1%]
  spare36 : INT ;
  spare38 : INT ;
  Snd : STRUCT
   PKW : STRUCT
    PKE : INT ;	//Logical Address Parameter
    Cmd : STRUCT
     spare : BYTE ;
     Read : BOOL ;
     Write : BOOL ;
    END_STRUCT ;
    PWE : DINT ;
   END_STRUCT ;
   Cmd : STRUCT
    Halt : BOOL ;
    Reserved9 : BOOL ;
    Reserved10 : BOOL ;
    DirectionRev : BOOL ;
    MultiMotorCfg1 : BOOL ;	//Use MultiMotor configuration 1
    MultiMotorCfg2 : BOOL ;	//Use MultiMotor configuration 2
    Spare14 : BOOL ;
    Spare15 : BOOL ;
    SwitchOn : BOOL ;
    EnableVoltage : BOOL ;
    QuickStop : BOOL ;
    EnableOperation : BOOL ;
    Reserved4 : BOOL ;
    Reserved5 : BOOL ;
    Reserved6 : BOOL ;
    FaultReset : BOOL ;
   END_STRUCT ;
   Speed : INT ;	//Target Speed e.g (LFR Logical Address 8502) [0.1Hz]
   PCD3 : INT ;
   PCD4 : INT ;
   PCD5 : INT ;
   PCD6 : INT ;
   PCD7 : INT ;
   PCD8 : INT ;
  END_STRUCT ;
  Rcv : STRUCT
   PKW : STRUCT
    PKE : INT ;	//Logical Address Parameter
    RWN : INT ;	//Code Answer
    PWE : DINT ;	//Paramter Value or Error reason
   END_STRUCT ;
   Status : STRUCT
    Reserved8 : BOOL ;
    Remote : BOOL ;
    TargetReached : BOOL ;
    InternalLimitActive : BOOL ;
    Reserved12 : BOOL ;
    Reserved13 : BOOL ;
    StopViaStopKey : BOOL ;
    DirectionRev : BOOL ;
    ReadySwitchOn : BOOL ;
    SwitchedOn : BOOL ;
    OperationEnabled : BOOL ;
    Fault : BOOL ;
    VoltageEnabled : BOOL ;
    QuickStop : BOOL ;
    SwitchedOnDisabled : BOOL ;
    Warning : BOOL ;
   END_STRUCT ;
   Speed : INT ;	//Actual Speed e.g (RFR Logical Address 3202) [0.1Hz]
   MultiMotorCfg : INT ;	//Active MultiMotor Configuration [0..2] (CNSF Logical Address 8020)
   PZD4 : INT ;
   PZD5 : INT ;
   PZD6 : INT ;
   PZD7 : INT ;
   PZD8 : INT ;
  END_STRUCT ;
  Par : STRUCT
   ParObjectNo : INT ;	//Is used for communication with PC, e.g. for message
   ParMsgType : INT ;	//Is used for message (translation of state)
   ParHornCode : INT ;	//Is used by horn module
   ParLogOff : BOOL ;	//Report is off
   ParManual : BOOL ;	//Manual mode without interlocking
   ParRestartDelay : BOOL ;	//No restart possible in StStopping
   ParHeavyStartup : BOOL ;	//Element with heavy startup
   ParStartwarning : BOOL ;
   ParValueAsUnit : BOOL ;	//Speed values as units not as not procent value
   ParIOByteNo : INT ;	//PROFIBUS: Address of first input and output byte
   ParMonTime : INT ;	//[0.1 s] After this time outputs must be equal inputs
   ParStartDelay : INT ;	//[0.1 s] Requested start delay time
   ParStartingTime : INT ;	//[0.1 s] Delay time, until the element is ready to start production
   ParStoppingTime : INT ;	//[0.1 s] Delay time, until the element has come to a standstill
   ParIdlingTime : INT ;	//[0.1 s] Requested idling time to stop element in automatic mode
   ParDelayFaultTime : INT ;	//[0.1 s] Requested fault delay time by negative flag of input
   ParDPNode1 : INT ;
   ParDPNode2 : INT ;
   ParUnitsBy100 : INT ;	//Unit by 100%
   OutMonTime : INT ;	//Actual time: Monitoring
   OutTransitionTime : INT ;	//Actual time: Starting, stopping, change direction, idling
   OutDelayFaultTime : INT ;	//Actual time: DelayTime
   OutStartDelay : INT ;
   InOutManPulseLen : INT ;	//Pulse length to start a the motor
   spare : DINT ;
  END_STRUCT ;
END_VAR
VAR_TEMP
  tmpLOGvalue : WORD ;	//LOG value
  tmpReport : BOOL ;	//Global LOG all
  tmpEnableRev : BOOL ;	//Global enable reverse
  tmpEnableFwd : BOOL ;	//Global enable forward
  tmpEnable : BOOL ;	//Global enable
  tmpDelayOver : BOOL ;	//Delay time is over
  tmpMonOver : BOOL ;	//Monitoring time is over
  tmpInpFault : BOOL ;	//Fault variable
  tmpHeavyStartup : BOOL ;	//Any element is starting with HeavyStartup
  tmpLocal : BOOL ;
  tmpStarted : BOOL ;
  tmpDPFaultInp : BOOL ;
  tmpDPFaultOutp : BOOL ;
  tmpLenDyn : INT ;	//Global enable forward
  tmpAddr : WORD ;
  tmpReturn : INT ;
  tmpAddrIO : DWORD ;
  tmpAddrRcv : DWORD ;
  tmpAddrSnd : DWORD ;
  tmpRunning : BOOL ;
  tmpFaultDelayRunning : BOOL ;
  tmpMultiMotorCfgTar : INT ;	//Target Multi Motor Config
END_VAR
BEGIN
NETWORK
TITLE =
      L     130;
      T     #tmpLenDyn;	//--> Len dynamic data in byte
      L     P##Rcv;
      L     DW#16#FFFFFF;
      AD;
      TAR2;
      +D;
      T     #tmpAddrRcv;
      L     P##Snd;
      L     DW#16#FFFFFF;
      AD;
      TAR2;
      +D;
      T     #tmpAddrSnd;
      L     #Par.ParIOByteNo;
      SLD   3;
      T     #tmpAddrIO;
NETWORK
TITLE = PC Control
//=== Test Object number =====================
      L     "SYS_DirectCtrlDB".PC.ObjectNo;	//PCControl.ObjectNo
      L     #Par.ParObjectNo;	//Input ObjectNo
      <>I;
      JC    Ctrl;
//=== Test OType      ========================
      L     1018;	//Input object type
      L     "SYS_DirectCtrlDB".PC.ObjectType;	//PCControl.ObjectType
      <>I;
      JC    Ctrl;
//=== Test Handshake =========================
      A     "SYS_DirectCtrlDB".PC.Hsk.FExamine;	// Handshake.FExamine
      JC    pExa;
      A     "SYS_DirectCtrlDB".PC.Hsk.FDefineCmd;	// Handshake.FDefineCmd
      O     "SYS_DirectCtrlDB".PC.Hsk.FDefineValue;	//Handshake.FDefineValue
      JC    pCmd;
      A     "SYS_DirectCtrlDB".PC.Hsk.FDefinePara;	// Handshake.FDefinePara
      JC    pPar;
pIni: L     2;	// FcInit
      UC    "SYS_DirectCtrl";
      JU    Ctrl;
// Write parameter 
pPar: L     "SYS_DirectCtrlDB".PC.Value[11];
      T     #Par.ParMonTime;
      L     "SYS_DirectCtrlDB".PC.Value[12];
      T     #Par.ParStartDelay;
      L     "SYS_DirectCtrlDB".PC.Value[13];
      T     #Par.ParStartingTime;
      L     "SYS_DirectCtrlDB".PC.Value[14];
      T     #Par.ParStoppingTime;
      L     "SYS_DirectCtrlDB".PC.Value[15];
      T     #Par.ParIdlingTime;
      L     "SYS_DirectCtrlDB".PC.Value[16];
      T     #Par.ParDelayFaultTime;
// Write new commands from PC to Interface object
pCmd: A     "SYS_DirectCtrlDB".PC.Cmd1[7];	// CmdManRevOn;
      AN    "GCS7_Gr_OutManualOff";	//Global.OutManualOff  [2.10]
      S     #InOutManRev;
      A     "SYS_DirectCtrlDB".PC.Cmd1[8];	// CmdOff
      AN    "GCS7_Gr_OutManualOff";	//Global.OutManualOff  [2.10]
      S     #CmdOff;
      A     "SYS_DirectCtrlDB".PC.Cmd1[9];	// CmdOn
      AN    "GCS7_Gr_OutManualOff";	//Global.OutManualOff  [2.10]
      S     #CmdOn;
      A     "SYS_DirectCtrlDB".PC.Cmd1[10];	// CmdNext
      S     #CmdNext;
      A     "SYS_DirectCtrlDB".PC.Cmd1[11];	// CmdFaultReset
      S     #CmdFaultReset;
      A     "SYS_DirectCtrlDB".PC.Cmd1[13];	// CmdManualOn
      S     #InManual;
      A     "SYS_DirectCtrlDB".PC.Cmd1[14];	// CmdReportOn
      S     #InReport;
      A     "SYS_DirectCtrlDB".PC.Cmd2[7];	// CmdManRevOff;
      R     #InOutManRev;
      A     "SYS_DirectCtrlDB".PC.Cmd2[13];	// CmdManualOff
      R     #InManual;
      A     "SYS_DirectCtrlDB".PC.Cmd2[14];	// CmdReportOff
      R     #InReport;
      AN    "SYS_DirectCtrlDB".PC.Cmd1[1];	// CmdOnTickFwd
      O     "GCS7_Gr_OutManualOff";	//Global.OutManualOff
      JC    pJ1;
      L     "SYS_DirectCtrlDB".PC.Cmd3;	// "SYS_PCControl".PC.Cmd3
      T     #Par.InOutManPulseLen;
//Define Value
pJ1:  AN    "SYS_DirectCtrlDB".PC.Hsk.FDefineValue;	// PC.Hsk.FDefineValue
      ON    #InManual;
      JC    pIni;
      L     "SYS_DirectCtrlDB".PC.Value[1];
      ITD;
      DTR;
      T     #InSpeed;
      JU    pIni;
pExa: L     #Par.ParMonTime;
      T     "SYS_DirectCtrlDB".PC.Value[11];
      L     #Par.ParStartDelay;
      T     "SYS_DirectCtrlDB".PC.Value[12];
      L     #Par.ParStartingTime;
      T     "SYS_DirectCtrlDB".PC.Value[13];
      L     #Par.ParStoppingTime;
      T     "SYS_DirectCtrlDB".PC.Value[14];
      L     #Par.ParIdlingTime;
      T     "SYS_DirectCtrlDB".PC.Value[15];
      L     #Par.ParDelayFaultTime;
      T     "SYS_DirectCtrlDB".PC.Value[16];
      TAR2;	// Address Dynamic datas
      T     "SYS_DirectCtrlDB".GC.InDynAddr;	// -->PCControl.GC.InDynAddr
      L     #tmpLenDyn;	// Length Dynamic datas
      T     "SYS_DirectCtrlDB".GC.InDynLen;	// -->PCControl.GC.InDynLen
      L     0;
      T     "SYS_DirectCtrlDB".GC.InParaAddr;	// -->PCControl.GC.InParaAddr
      T     "SYS_DirectCtrlDB".GC.InParaLen;	// -->PCControl.GC.InParaLen
      L     10;	//Revision
      T     "SYS_DirectCtrlDB".GC.Revision;
      L     DINO;
      T     "SYS_DirectCtrlDB".GC.InDBNr;
      JU    pIni;
Ctrl: NOP   0;
NETWORK
TITLE = (Profibus) Read data and store Data 
      L     #Par.ParIOByteNo;
      T     #tmpAddr;
      A     #InSimulation;
      JC    rSim;
      CALL  "SIEMENS_DPRD_DAT" (
           LADDR                    := #tmpAddr,
           RET_VAL                  := #tmpReturn,
           RECORD                   := #Rcv.PKW);
      L     #tmpReturn;
      L     0;
      <>I;
      =     #OutComFaultRead;
      LAR1  #tmpAddrIO;
      L     PIW [AR1,P#8.0];
      LAR1  #tmpAddrRcv;
      T     DIW [AR1,P#8.0];
      LAR1  #tmpAddrIO;
      L     PIW [AR1,P#10.0];
      LAR1  #tmpAddrRcv;
      T     DIW [AR1,P#10.0];
      LAR1  #tmpAddrIO;
      L     PIW [AR1,P#12.0];
      LAR1  #tmpAddrRcv;
      T     DIW [AR1,P#12.0];
      LAR1  #tmpAddrIO;
      L     PIW [AR1,P#14.0];
      LAR1  #tmpAddrRcv;
      T     DIW [AR1,P#14.0];
      LAR1  #tmpAddrIO;	//[1.5]
      L     PIW [AR1,P#16.0];	//[1.5]
      LAR1  #tmpAddrRcv;	//[1.5]
      T     DIW [AR1,P#16.0];	//[1.5]
      LAR1  #tmpAddrIO;	//[1.5]
      L     PIW [AR1,P#18.0];	//[1.5]
      LAR1  #tmpAddrRcv;	//[1.5]
      T     DIW [AR1,P#18.0];	//[1.5]
      LAR1  #tmpAddrIO;	//[1.5]
      L     PIW [AR1,P#20.0];	//[1.5]                                                  
      LAR1  #tmpAddrRcv;	//[1.5]
      T     DIW [AR1,P#20.0];	//[1.5]
      LAR1  #tmpAddrIO;	//[1.5]
      L     PIW [AR1,P#22.0];	//[1.5]
      LAR1  #tmpAddrRcv;	//[1.5]
      T     DIW [AR1,P#22.0];	//[1.5]
      JU    rDP;
//read from Simulation
rSim: R     #OutComFaultRead;
      A     "GCS7_Gr_SimDPtoImage";
      L     P#I 0.0;
      JC    rDB1;
      OPN   "TEST_IOSimuliInput";
      L     P#DBX 0.0;
rDB1: L     #Par.ParIOByteNo;
      SLD   3;
      +D;
      T     #tmpAddrIO;
      LAR1  #tmpAddrIO;
      L     D [AR1,P#0.0];
      LAR1  #tmpAddrRcv;
      T     DID [AR1,P#0.0];
      LAR1  #tmpAddrIO;
      L     D [AR1,P#4.0];
      LAR1  #tmpAddrRcv;
      T     DID [AR1,P#4.0];
      LAR1  #tmpAddrIO;
      L     D [AR1,P#8.0];
      LAR1  #tmpAddrRcv;
      T     DID [AR1,P#8.0];
      LAR1  #tmpAddrIO;	//[1.5]
      L     D [AR1,P#12.0];	//[1.5]
      LAR1  #tmpAddrRcv;	//[1.5]
      T     DID [AR1,P#12.0];	//[1.5]
      LAR1  #tmpAddrIO;	//[1.5]
      L     D [AR1,P#16.0];	//[1.5]
      LAR1  #tmpAddrRcv;	//[1.5]
      T     DID [AR1,P#16.0];	//[1.5]
      LAR1  #tmpAddrIO;	//[1.5]
      L     D [AR1,P#20.0];	//[1.5]
      LAR1  #tmpAddrRcv;	//[1.5]
      T     DID [AR1,P#20.0];	//[1.5]
rDP:  NOP   0;
//===============================
//LC Parameter 
//===============================
      L     "SYS_DirectCtrlLCDB".PC.ObjectNo;
      L     #Par.ParObjectNo;
      <>I;
      JC    rJ0;
//-------------------------------------------
//Check Answer Examine
      ON    "SYS_DirectCtrlLCDB".PC.Hsk.FExamine;
      ON    #Snd.PKW.Cmd.Read;
      JC    rW1;
      L     #Rcv.PKW.PKE;
      L     #Snd.PKW.PKE;
      ==I;
      JCN   rW1;
      L     #Rcv.PKW.RWN;
      L     1;
      ==I;
      JCN   rW1;
      R     #Snd.PKW.Cmd.Read;
      T     "SYS_DirectCtrlLCDB".PC.Value[2];
      L     #Rcv.PKW.PWE;
      SRD   16;
      T     "SYS_DirectCtrlLCDB".PC.Value[3];
      L     #Rcv.PKW.PWE;
      T     "SYS_DirectCtrlLCDB".PC.Value[4];
      L     12;
      CALL  "SYS_DirectCtrl";
      JU    rJ1;
//-------------------------------------------
//Check Answer Write
rW1:  AN    "SYS_DirectCtrlLCDB".PC.Hsk.FDefinePara;
      ON    #Snd.PKW.Cmd.Write;
      JC    rJ1;
      L     #Rcv.PKW.PKE;
      L     #Snd.PKW.PKE;
      ==I;
      JCN   rJ1;
      L     #Rcv.PKW.RWN;
      L     2;
      ==I;
      JC    rWA1;
      L     #Rcv.PKW.RWN;
      L     7;
      ==I;
      JC    rWA1;
      JU    rJ1;
rWA1: R     #Snd.PKW.Cmd.Write;
      L     #Rcv.PKW.RWN;
      T     "SYS_DirectCtrlLCDB".PC.Value[2];
      L     12;
      CALL  "SYS_DirectCtrl";
      JU    rJ1;
//-------------------------------------------
//Examine Parameter
rJ1:  AN    "SYS_DirectCtrlLCDB".PC.Hsk.FExamine;
      JC    rJ2;
      O     #Snd.PKW.Cmd.Read;
      O     #Snd.PKW.Cmd.Write;
      JC    rJ2;
      S     #Snd.PKW.Cmd.Read;
      L     "SYS_DirectCtrlLCDB".PC.Value[1];
      T     #Snd.PKW.PKE;
      JU    rJ9;
//-------------------------------------------
//Write Parameter
rJ2:  AN    "SYS_DirectCtrlLCDB".PC.Hsk.FDefinePara;
      JC    rJ0;
      O     #Snd.PKW.Cmd.Read;
      O     #Snd.PKW.Cmd.Write;
      JC    rJ0;
      S     #Snd.PKW.Cmd.Write;
      L     "SYS_DirectCtrlLCDB".PC.Value[1];
      T     #Snd.PKW.PKE;
      L     "SYS_DirectCtrlLCDB".PC.Value[3];
      SLD   16;
      L     "SYS_DirectCtrlLCDB".PC.Value[4];
      OD;
      T     #Snd.PKW.PWE;
      JU    rJ9;
//===============================
//Init Flag
//===============================
rJ0:  L     #Rcv.PKW.PKE;
      L     #Snd.PKW.PKE;
      <>I;
      JC    rJ9;
      L     #Rcv.PKW.RWN;
      L     1;
      ==I;
      R     #Snd.PKW.Cmd.Read;
      L     #Rcv.PKW.RWN;
      L     2;
      ==I;
      A(;
      L     #Snd.PKW.PWE;
      L     #Rcv.PKW.PWE;
      ==I;
      );
      O(;
      L     #Rcv.PKW.RWN;
      L     7;
      ==I;
      );
      R     #Snd.PKW.Cmd.Write;
rJ9:  NOP   0;
NETWORK
TITLE = DPFault
      A     #InDPFault;
      =     #OutDPFault;
NETWORK
TITLE = Multi Motor Configuration
      A     #InMultiMotorCfg0;	//[1.3]
      L     1;	//[1.3] Return Value of MultiMotorCfg 0 is 1
      JC    MCJ1;	//[1.3]
      A     #InMultiMotorCfg1;	//[1.3]
      L     2;	//[1.3] Return Value of MultiMotorCfg 1 is 2
      JC    MCJ1;	//[1.3]
      A     #InMultiMotorCfg2;	//[1.3]
      L     3;	//[1.3] Return Value of MultiMotorCfg 2 is 3
      JC    MCJ1;	//[1.3]
      L     0;	//[1.3]
MCJ1: T     #tmpMultiMotorCfgTar;	//[1.3]
      L     2;	//[1.3]
      L     #tmpMultiMotorCfgTar;	//[1.3]
      ==I;	//[1.3]
      =     #Snd.Cmd.MultiMotorCfg1;	//[1.3]
      L     3;	//[1.3]
      L     #tmpMultiMotorCfgTar;	//[1.3]
      ==I;	//[1.3]
      =     #Snd.Cmd.MultiMotorCfg2;	//[1.3]
NETWORK
TITLE =  All State Init
      NOP   0;
//===Global Group Orders===
      A     "GCS7_Gr_OutManualOff";	//Global.OutManualOff
      R     #InManual;
      AN    #InManual;
      A     #InLocal;
      =     #tmpLocal;
//Force Off
//   U     "GCS7_Gr_OutForceOff"
//   R     #InForce
//[1.5]->Begin
//-Fault reset---
      A     "GCS7_Gr_OutFaultReset";
      S     #CmdFaultReset;
//[1.5]<-End
//---Report is on---
      O     "GCS7_Gr_OutReportAll";	//---Global OutReportAll
      O     #InReport;
      =     #tmpReport;
//---Heavy Startup---
      A     "GCS7_Gr_InHeavyStartup";	//---Global InHeavyStartup
      A     #Par.ParHeavyStartup;
      =     #tmpHeavyStartup;
//===Global Enable
      A     #CmdOff;
      R     #CmdOn;
      R     #CmdNext;
//---Enable / Manual No Interlocking Mode---
      AN    #InManual;
      JC    AUT;
      A(;
      A     #InEnableFwd;
      AN    #Par.ParManual;
      O;
      AN    #InOutManRev;
      A     #Par.ParManual;
      );
      AN    #InHWStop;
      AN    #OutDPFault;
      =     #tmpEnableFwd;
      A(;
      A     #InEnableRev;
      AN    #Par.ParManual;
      O;
      A     #InOutManRev;
      A     #Par.ParManual;
      );
      AN    #InHWStop;
      AN    #OutDPFault;
      =     #tmpEnableRev;
      JU    ENAB;
//---Enable / Automatic Interlocking Mode---
AUT:  A     #InEnableFwd;
      AN    #InHWStop;
      AN    #OutDPFault;
      AN    #InLocal;
      =     #tmpEnableFwd;
      A     #InEnableRev;
      AN    #InHWStop;
      AN    #OutDPFault;
      AN    #InLocal;
      =     #tmpEnableRev;
//---Enable / HardwareStop---
ENAB: X     #tmpEnableFwd;	//---Global Enable
      X     #tmpEnableRev;
      A(;	//[1.3]
      L     #Rcv.MultiMotorCfg;	//[1.3]
      L     #tmpMultiMotorCfgTar;	//[1.3]
      ==I;	//[1.3]
      O(;	//[1.3]
      L     0;	//[1.3]
      ==I;	//[1.3]
      );	//[1.3]
      );	//[1.3]
      =     #tmpEnable;
//---Both Inputs or InpFaultDevice active
      A     #InpOverload;
      O     #InpIsolated;
      O     #InpService;
      AN    #StStopped;
      AN    #StFault;
      O     #OutComFaultRead;
      O     #OutComFaultWrite;
      O     #Rcv.Status.Fault;
      AN    #InForce;
      =     #tmpInpFault;
//---Test Started ---------------
      O     #StStartedFwd;
      O     #StStartedRev;
      =     #tmpStarted;
//---Test Running 
      A     #Rcv.Status.OperationEnabled;
      A     #InpContactor;
      =     #tmpRunning;
NETWORK
TITLE = Start as Pulse
      AN    #tmpEnable;
      ON    #InManual;
      O     #CmdOff;
      JC    STP1;
      L     0;
      L     #Par.InOutManPulseLen;
      >=I;
      JC    STP2;
      A     #StStopped;
      AN    #OutStartRequestMan;
      S     #CmdOn;
      ON    "GCS7_Gr_OutTick200ms";	// Decrement all 200ms
      O     #OutStartRequestMan;	//[5.0]
      JC    STP2;
      +     -2;
      T     #Par.InOutManPulseLen;
      L     0;
      >I;
      JC    STP2;
      S     #CmdOff;
STP1: L     0;
      T     #Par.InOutManPulseLen;
STP2: NOP   0;
NETWORK
TITLE = Fault delay time: ParDelayTime 
//Test or Running delay time ====================
//---Condition for Delay Fault
      A     #StStartedFwd;
      O     #StStartedRev;
      A     #Snd.Cmd.EnableOperation;
      AN    #Rcv.Status.OperationEnabled;
      JC    TFF1;
      R     #tmpFaultDelayRunning;
      L     #Par.ParDelayFaultTime;
      T     #Par.OutDelayFaultTime;
      JU    TFF0;
TFF1: AN    "GCS7_Gr_OutTick200ms";	// Decrement all 200ms
      L     #Par.OutDelayFaultTime;
      JC    TFF3;
      +     -2;
TFF3: T     #Par.OutDelayFaultTime;
      L     0;
      >I;
      =     #tmpFaultDelayRunning;
      JC    TFF0;
      T     #Par.OutDelayFaultTime;
TFF0: NOP   0;
NETWORK
TITLE = Start Request //[5.0]
      NOP   0;
//--------------
      A     #CmdNext;
      O     #CmdOn;
      O     #OutStartRequestAuto;
      AN    #CmdOff;
      A     #tmpEnable;
      AN    #InManual;
      AN    #InSeqStop;
      A(;
      A     #StStopped;
      O     #StStopping;
      );
      =     #OutStartRequestAuto;
//--------------
      A     #CmdOn;
      O     #OutStartRequestMan;
      AN    #CmdOff;
      A     #tmpEnable;
      A     #InManual;
      A     #StStopped;
      =     #OutStartRequestMan;
NETWORK
TITLE = Start-Delay //[5.0]
      A     #OutStartRequestAuto;
      JC    SDY1;
      L     #Par.ParStartDelay;
      T     #Par.OutStartDelay;
SDY1: L     0;
      L     #Par.OutStartDelay;
      <I;
      A     #OutStartRequestAuto;
      =     #OutStartDelay;
      JCN   SDY2;
      AN    "GCS7_Gr_OutTick200ms";
      JC    SDY2;
      L     #Par.OutStartDelay;
      +     -2;
      T     #Par.OutStartDelay;
SDY2: NOP   0;
NETWORK
TITLE = Startwarning  
NETWORK
TITLE = States
      A     #StStopped;	//===State machine===
      JC    S0;
      O     #StStartedFwd;
      O     #StStartedRev;
      JC    S2;
      A     #StStopping;
      JC    S3;
      A     #StStarting;
      JC    S1;
      A     #StFault;
      JC    S4;
      S     #StStopped;	//Initialise: goto StStopped
      JU    S0;
NETWORK
TITLE = StStopped
      NOP   0;
//Transiiton to StStopped
xxS0: R     #StStopping;
      S     #StStopped;
      JU    LOG1;
//==============================
//State
//==============================
//---Condition for StFault
S0:   A     #tmpInpFault;
      AN    #tmpLocal;
      JC    xxS4;
//---Condition for StStarting
      A(;
      A     #OutStartRequestAuto;
      AN    #OutStartDelay;
      O     #OutStartRequestMan;
      AN    #tmpHeavyStartup;
      AN    #OutStartWarning;
      AN    #tmpLocal;
      O;
      A     #tmpLocal;
      A     #Rcv.Status.OperationEnabled;
      );
      JC    xxS1;
      JU    SAVE;
NETWORK
TITLE = StStarting
      NOP   0;
//==============================
// Any transition to StStarting
//==============================
xxS1: SET;
      R     #StStopped;
      R     #StStopping;
      S     #StStarting;
      L     #Par.ParMonTime;	// Set actual vaule of timer
      T     #Par.OutMonTime;
      L     #Par.ParStartingTime;
      T     #Par.OutTransitionTime;
      A     #Par.ParHeavyStartup;
      S     "GCS7_Gr_InHeavyStartup";
// Maintanance Counter Startups
      L     #OutCntStartup;
      +     L#1;
      T     #OutCntStartup;
      JU    SAVE;
//==============================
//State
//==============================
//---Condition for StFault
S1:   A     #tmpInpFault;
      AN    #tmpLocal;
      JC    S1S4;
//---Condition for StStopped
      AN    #tmpEnable;
      O     #CmdOff;
      AN    #tmpLocal;
      O;
      A     #InSeqStop;
      AN    #InManual;
      AN    #tmpLocal;
      O;
      AN    #Rcv.Status.OperationEnabled;
      A     #tmpLocal;
      JC    S1S3;
//---Condition for StStarting
      AN    "GCS7_Gr_OutTick200ms";
      L     #Par.OutTransitionTime;	// Set Timer 
      JC    S13;
      L     #Par.OutMonTime;
      +     -2;
      T     #Par.OutMonTime;
      L     #Par.OutTransitionTime;
      +     -2;
      T     #Par.OutTransitionTime;
S13:  L     0;
      <=I;
      =     #tmpDelayOver;	// Starting time over
//---Condition for StStarted
      A     #tmpRunning;
      O     #InForce;
      A     #tmpDelayOver;
      JC    xxS2;
//---Condition for StFault
      L     #Par.OutMonTime;
      L     0;	// Monitoring time over
      <=I;
      AN    #tmpLocal;
      AN    #tmpRunning;
      JC    S1S4;
      JU    SAVE;
//---Transition -> StStopping
S1S3: R     #StStarting;
      A     #tmpHeavyStartup;	// Clear Global InHeavyStartup
      R     "GCS7_Gr_InHeavyStartup";
      JU    xxS3;
//---Transition -> StFault
S1S4: R     #StStarting;
      A     #tmpHeavyStartup;	// Clear Global InHeavyStartup
      R     "GCS7_Gr_InHeavyStartup";
      JU    xxS4;
NETWORK
TITLE = StStarted
      NOP   0;
//---Transition -> StStartedXxx
xxS2: SET;
      R     #StStarting;
      L     0;
      T     #Par.OutMonTime;
      T     #Par.OutTransitionTime;
      A     #tmpHeavyStartup;	// Clear Global InHeavyStartup
      R     "GCS7_Gr_InHeavyStartup";
//---Transition -> StStartedFwd
      AN    #Rcv.Status.DirectionRev;
      AN    #InForce;
      O;
      A     #tmpEnableFwd;
      A     #InForce;
      S     #StStartedFwd;
      R     #StStartedRev;
      JC    LOG1;
//---Transition -> StStartedRev
      S     #StStartedRev;
      R     #StStartedFwd;
      JU    LOG1;
//==============================
//State
//==============================
//---Condition for Stopping when Change Direction
S2:   A     #tmpEnableRev;
      A     #StStartedFwd;
      AN    #tmpLocal;
      O;
      A     #tmpEnableFwd;
      A     #StStartedRev;
      AN    #tmpLocal;
      JC    xxS3;
//---Condition for StFault
      A(;
      AN    #tmpRunning;
      AN    #tmpFaultDelayRunning;
      AN    #InForce;
      A     #Snd.Cmd.EnableOperation;
      O     #tmpInpFault;
      O;
      AN    #InpContactor;
      AN    #InForce;
      );
      AN    #tmpLocal;
      JC    xxS4;
//Change Direction
      AN    #Rcv.Status.DirectionRev;
      A     #Snd.Cmd.EnableOperation;
      A     #StStartedRev;
      JC    xxS2;
      A     #Rcv.Status.DirectionRev;
      A     #Snd.Cmd.EnableOperation;
      A     #StStartedFwd;
      JC    xxS2;
// Maintanance Counter
      AN    "GCS7_Gr_OutTick1s";	// Increment all s
      JC    S2MT;
      L     #OutTimeStarted;
      +     L#1;
      T     #OutTimeStarted;
//===Local Mode======================
S2MT: AN    #tmpLocal;
      JC    S2J1;
//---Condition for StStopping: local mode
      AN    #Rcv.Status.OperationEnabled;
      AN    #tmpFaultDelayRunning;
      JC    xxS3;
      JU    SAVE;
//===Automatic Mode======================
//---Condition for StStopping: autmatic
S2J1: AN    #tmpEnable;	// other modes
      O     #CmdOff;
      O;
      AN    #Rcv.Status.OperationEnabled;
      AN    #tmpFaultDelayRunning;
      AN    #InForce;
      JC    xxS3;
//---Idling time ----------------------
      A     #InSeqStop;
      A     #OutIdling;
      JC    S2I1;
      L     #Par.ParIdlingTime;
      T     #Par.OutTransitionTime;
      A     #InSeqStop;
      AN    #InManual;
      S     #OutIdling;
      JU    SAVE;
S2I1: AN    "GCS7_Gr_OutTick200ms";
      L     #Par.OutTransitionTime;
      JC    S2I3;
      +     -2;
      T     #Par.OutTransitionTime;
S2I3: L     0;
      <=I;	// Idling time over
      JC    xxS3;	//--> StStopping
      JU    SAVE;
NETWORK
TITLE = StStopping
      NOP   0;
//=============================
//Any transition to StStopping
//=============================
xxS3: SET;
      S     #StStopping;
      R     #OutIdling;
      R     #StStartedFwd;
      R     #StStartedRev;
      L     #Par.ParMonTime;	// Set monitoring time
      T     #Par.OutMonTime;
      L     #Par.ParStoppingTime;	// Set stopping time
      T     #Par.OutTransitionTime;
      JU    SAVE;
//==============================
//State
//==============================
//---Condition for StFault
S3:   A     #tmpInpFault;
      AN    #tmpLocal;
      JC    xxS4;
//---Condition for StStarting in InLocal
      AN    #tmpInpFault;
      A     #Rcv.Status.OperationEnabled;	//[1.1]
      A     #tmpLocal;
      JC    xxS1;
//---Condition for StStarting: no Restart
      A     #Par.ParRestartDelay;
      O     #tmpHeavyStartup;
      JC    S3J2;
      A     #OutStartRequestAuto;
      AN    #OutStartDelay;
      O     #OutStartRequestMan;
      AN    #tmpHeavyStartup;
      AN    #OutStartWarning;
      JC    xxS1;
//---Condition for StStopping
S3J2: AN    "GCS7_Gr_OutTick200ms";
      L     #Par.OutTransitionTime;	// Set Timer 
      JC    S3J3;
      L     #Par.OutMonTime;	//---Condition for StStopped
      +     -2;	// Set actual timer
      T     #Par.OutMonTime;
      L     #Par.OutTransitionTime;
      +     -2;
      T     #Par.OutTransitionTime;
S3J3: L     0;
      <=I;	// Stopping time over
      =     #tmpDelayOver;
//---Condition for StStopped
      A     #tmpDelayOver;	// Stopped
      AN    #Rcv.Status.OperationEnabled;
      JC    xxS0;
//Monitoring Time
      L     #Par.OutMonTime;
      L     0;	// Monitoring time over
      <=I;
      =     #tmpMonOver;
      AN    #tmpMonOver;
      ON    #tmpDelayOver;	// Stopping time over
      JC    SAVE;
//---Transtition -> StFault
      JU    xxS4;
NETWORK
TITLE =  StFault
      NOP   0;
//==============================
// Any transiton to Fault  
//==============================
xxS4: SET;
      R     #tmpEnable;
      R     #StStopped;
      R     #StStopping;
      R     #StStartedFwd;
      R     #StStartedRev;
      R     #OutDelayFault;
      R     #OutIdling;
// Maintanance Counter Faults
      A     #StFault;
      JC    S4T2;
      L     #OutCntFault;
      +     L#1;
      T     #OutCntFault;
S4T2: SET;
      S     #StFault;
      S     "GCS7_Gr_InFaultFlag";	// Global.InFaultFlag
//    S     #tmpTimeClear               // Reset actual timer value
      CALL  "SYS_Horn_Code" (
           FcCode                   := 1,
           ParObjectType            := 1018,
           ParObjectNo              := #Par.ParObjectNo,
           ParHornCode              := #Par.ParHornCode);
      L     0;
      T     #Par.OutMonTime;
      L     #Par.ParStoppingTime;
      T     #Par.OutTransitionTime;
      SET;
S4S4: JU    LOG4;
//==============================
//State
//==============================
// Maintanance Counter Fault Time
S4:   AN    "GCS7_Gr_OutTick1s";	// Increment all s
      JC    S4MT;
      L     #OutTimeFaulted;
      +     L#1;
      T     #OutTimeFaulted;
//===logic
S4MT: L     0;	//---Condition to count stopping time
      L     #Par.OutTransitionTime;	// Set Timer 
      >=I;
      ON    "GCS7_Gr_OutTick200ms";
      JC    S4J1;
      +     -2;
      T     #Par.OutTransitionTime;
//Set Timer Fault Reset
S4J1: AN    #CmdFaultReset;	//[1.6]
      AN    "GCS7_Gr_OutFaultReset";	//[1.6]
      JC    S4D1;	//[1.6]
      L     30;	//[1.6]
      T     #Par.OutMonTime;	//[1.6]
//---Condition for StFault
S4D1: L     0;	//[1.6]
      L     #Par.OutMonTime;	//[1.6]
      <>I;	//[1.6]
      O     #tmpLocal;	//[1.6]
      JC    S4D2;	//[1.6]  --> Run Timer Fault Reset
      A     #Rcv.Status.Fault;
      AN    #tmpLocal;
      AN    #OutFaultDev;
      JC    S4S4;
      JU    SAVE;	//[1.6]
//-- Run Timer Fault Reset              //[1.6]
S4D2: AN    "GCS7_Gr_OutTick200ms";	//[1.6]
      A     #Rcv.Status.Fault;	//[1.6]
      AN    #tmpLocal;	//[1.6]
      JC    SAVE;	//[1.6]
      L     #Par.OutMonTime;	//[1.6]
      +     -2;	//[1.6]
      T     #Par.OutMonTime;	//[1.6]
      L     0;	//[1.6]
      >I;	//[1.6]
      JC    SAVE;	//[1.6]
      T     #Par.OutMonTime;	//[1.6]
//---Condition for StFault with LOG
      A     #OutpContactor;
      AN    #InpContactor;
      O     #Rcv.Status.Fault;
      O     #InpIsolated;
      O     #InpOverload;
      O     #InpService;
      O     #tmpInpFault;	// MessageClass Error Fault stopping
      AN    #InForce;
      AN    #tmpLocal;
      JC    S4S4;
      R     #StFault;	//---Transition -> StStopping
      S     #StStopping;
      R     #OutIdling;
      L     #Par.ParMonTime;	// Set monitoring time
      T     #Par.OutMonTime;
      JU    LOG9;
NETWORK
TITLE = LOG Message
//LOG transition to StStopped,StStartedXxx
LOG1: AN    #tmpReport;	// ReportAll?
      JC    SAVE;
      A     #StStartedFwd;
      L     B#(4, 2);	// MessageClass Info started fwd
      JC    LOG;
      A     #StStartedRev;
      L     B#(4, 5);	// MessageClass Info started rev
      JC    LOG;
      A     #StStopped;
      L     B#(4, 0);	// MessageClass Info stopped
      JC    LOG;	// [4.2]
      JU    SAVE;
//LOG transition to fault
LOG4: O     #OutComFaultRead;	//[1.7]
      O     #OutComFaultWrite;	//[1.7]
      S     #OutFaultDev;	//[1.7]
      L     B#(1, 96);	//[1.7] MessageClass Error fault Profibus
      JC    LOG;	//[1.7]
      A     #Rcv.Status.Fault;
      S     #OutFaultDev;
      L     B#(1, 10);	// MessageClass Error fault device
      JC    LOG;
      A     #InpIsolated;
      S     #OutFaultIsolated;	//[5.0]
      L     B#(1, 14);	// MessageClass Error fault isolated
      JC    LOG;
      A     #InpOverload;
      S     #OutFaultOverload;	//[5.0]
      L     B#(1, 15);	// MessageClass Error fault Overload
      JC    LOG;
      A     #InpService;
      S     #OutFaultService;	//[5.0]
      L     B#(1, 16);	// MessageClass Error fault Service
      JC    LOG;
      AN    #Rcv.Status.Remote;
      L     B#(1, 18);	// MessageClass Error fault remote
      JC    LOG;
      A     #tmpStarted;
      L     B#(1, 11);	// MessageClass Error fault started
      JC    LOG;
      A     #OutpContactor;
      AN    #InpContactor;
      L     B#(1, 17);	// MessageClass Error fault contactor
      S     #OutFaultStarting;	//[5.0]
      JC    LOG;
      AN    #tmpEnable;	// Fault Stopping
      O     #OutFaultStopping;
      L     B#(1, 13);
      S     #OutFaultStopping;	//[5.0]
      JC    LOG;
      L     B#(1, 12);	// MessageClass Error fault starting
      S     #OutFaultStarting;	//[5.0]
      JU    LOG;
//Log fault cancelled
LOG9: L     B#(3, 9);	// MessageClass Operater "fault cancelled"
LOG:  A     #Par.ParLogOff;	//---Set LOG Message
      JC    SAVE;
      T     #tmpLOGvalue;
      L     W#16#FF;
      AW;
      T     #OutAlarmNoLog;
      CALL  "GCS7_LogConvert" (
           ObjectNo                 := #Par.ParObjectNo,
           MsgType                  := #Par.ParMsgType,
           ClassMsgTxt              := #tmpLOGvalue,
           OType                    := 1018);	// LOG Message Converter / Entry / Contains Class and TextNo
NETWORK
TITLE = Reset Fault Flag
SAVE: AN    #StFault;
      R     #OutFaultStopping;
      R     #OutFaultStarting;
      R     #OutFaultOverload;
      R     #OutFaultIsolated;
      R     #OutFaultService;
      R     #OutFaultDev;
NETWORK
TITLE = State Code
      NOP   0;
//--Stopped, Substate ---
      AN    #StStopped;
      JC    STC2;
      L     41;	//Code: StStopped.HWStop
      A     #InHWStop;
      JC    STC9;
      L     51;	//Code: StStopped.DPFault
      A     #InDPFault;
      O     #OutComFaultRead;
      O     #OutComFaultWrite;
      JC    STC9;
      A     #Rcv.Status.Fault;
      L     30;	//Code: StStopped.InpFaultDev
      JC    STC9;
      A     #CmdNext;
      AN    #tmpLocal;
      L     9;	// Code: starting requested
      JC    STC9;
      L     1;	// Code: stopped
      JC    STC9;
//--------------------
STC2: A     #StStarting;
      L     2;	// Code: starting
      JC    STC9;
      A     #StStartedFwd;
      L     4;	// 2.6 Code: started forward
      JC    STC9;
//--------------------
      A     #StStartedRev;
      L     6;	// 2.6: Code: started reverse
      JC    STC9;
//--------------------
      A     #StStopping;
      L     7;	// Code: stopping
      JC    STC9;
      A     #Rcv.Status.Fault;	// Code: StFault.ATV
      L     31;	// 
      JC    STC9;	// 
      L     32;	// Code: fault
STC9: L     #StCode;	// Old state code
      TAK;
      T     #StCode;	// Save state code
      <>I;
      L     3;	// Load code for CBit methode
      CC    "SYS_CBitCtrl";
NETWORK
TITLE = Command FU /IO
      AN    #tmpLocal;
      =     #OutpContactor;
      AN    #tmpLocal;
      =     #Snd.Cmd.EnableVoltage;
      =     #Snd.Cmd.QuickStop;
//--------------
      A     #InPrestart;
      O     #tmpEnableFwd;
      O     #tmpEnableRev;
      AN    #tmpLocal;
      A     #Rcv.Status.ReadySwitchOn;
      =     #Snd.Cmd.SwitchOn;
//--------------
      A     #tmpEnableFwd;
      O     #tmpEnableRev;
      AN    #StStopped;
      AN    #StFault;
      AN    #StStopping;
      A     #Snd.Cmd.SwitchOn;
      A     #Rcv.Status.SwitchedOn;
      A(;
      A     #StStarting;
      O     #Snd.Cmd.EnableOperation;
      );
      A     #InpContactor;
      =     #Snd.Cmd.EnableOperation;
//--------------
      A     #tmpEnableFwd;
      R     #Snd.Cmd.DirectionRev;
      A     #tmpEnableRev;
      S     #Snd.Cmd.DirectionRev;
//--------------
      A     #CmdFaultReset;
      S     #Snd.Cmd.FaultReset;
      AN    #Rcv.Status.Fault;
      O     #tmpLocal;
      R     #Snd.Cmd.FaultReset;
//--------------
//Convert target value
      A     #Par.ParValueAsUnit;
      L     #InSpeed;
      JC    dpJ1;
      L     1.000000e+02;
      /R;
      L     #Par.ParUnitsBy100;
      DTR;
      *R;
      RND+;
      JU    dpJ2;
dpJ1: RND;
dpJ2: T     #Snd.Speed;
//--------------
//Convert actual value
      L     #Rcv.Speed;
      ITD;
      DTR;
      A     #Par.ParValueAsUnit;	//[1.8]
      JC    dpJ3;	//[1.8]
      L     #Par.ParUnitsBy100;
      DTR;
      /R;
      L     1.000000e+02;
      *R;
dpJ3: T     #OutSpeed;
NETWORK
TITLE = (Profibus) Send Data
      A     #InSimulation;
      JC    sSim;
      CALL  "SIEMENS_DPWR_DAT" (
           LADDR                    := #tmpAddr,
           RECORD                   := #Snd.PKW,
           RET_VAL                  := #tmpReturn);
      L     #tmpReturn;
      L     0;
      <>I;
      =     #OutComFaultWrite;
      LAR1  #tmpAddrSnd;
      L     DIW [AR1,P#8.0];
      LAR1  #tmpAddrIO;
      T     PQW [AR1,P#8.0];
      LAR1  #tmpAddrSnd;
      L     DIW [AR1,P#10.0];
      LAR1  #tmpAddrIO;
      T     PQW [AR1,P#10.0];
      LAR1  #tmpAddrSnd;
      L     DIW [AR1,P#12.0];
      LAR1  #tmpAddrIO;
      T     PQW [AR1,P#12.0];
      LAR1  #tmpAddrSnd;
      L     DIW [AR1,P#14.0];
      LAR1  #tmpAddrIO;
      T     PQW [AR1,P#14.0];
      JU    DP_C;
//write to Simulation
sSim: R     #OutComFaultWrite;
      A     "GCS7_Gr_SimDPtoImage";
      L     P#Q 0.0;
      JC    rDB2;
      OPN   "TEST_IOSimuliOutput";
      L     P#DBX 0.0;
rDB2: L     #Par.ParIOByteNo;
      SLD   3;
      +D;
      T     #tmpAddrIO;
      LAR1  #tmpAddrSnd;
      L     DID [AR1,P#0.0];
      LAR1  #tmpAddrIO;
      T     D [AR1,P#0.0];
      LAR1  #tmpAddrSnd;
      L     DID [AR1,P#4.0];
      LAR1  #tmpAddrIO;
      T     D [AR1,P#4.0];
      LAR1  #tmpAddrSnd;
      L     DIW [AR1,P#8.0];
      LAR1  #tmpAddrIO;
      T     W [AR1,P#8.0];
      LAR1  #tmpAddrSnd;
      L     DIW [AR1,P#10.0];
      LAR1  #tmpAddrIO;
      T     W [AR1,P#10.0];
DP_C: NOP   0;
NETWORK
TITLE = Global End
      CLR;	//---Clear all commands
      =     #CmdOn;
      =     #CmdOff;
      =     #CmdNext;
      =     #CmdFaultReset;
//-- Init Start Request
      AN    #OutStartDelay;
      AN    #OutStartWarning;
      R     #OutStartRequestAuto;
      R     #OutStartRequestMan;
//--Output for group 
      A     M 11.7;
      A     #InLocal;
      A     #InManual;
      O     #InForce;
      JC    ENJ2;
      A     #OutDPFault;
      S     "GCS7_Gr_InDPFault";
      A     #InHWStop;
      S     "GCS7_Gr_InHWStop";
ENJ2: NOP   0;
      A     #InForce;
      S     "GCS7_Gr_InForce";
      A     #InManual;
      S     "GCS7_Gr_InManual";
// No fault when not used element in manual mode
      AN    M 11.7;
      ON    #InLocal;
      A     #StFault;
      =     #OutFaultRelevant;
END_FUNCTION_BLOCK

